// Block: PPrgArchive10

DATA_BLOCK PPrgArchive10
VERSION : 0.1
   NON_RETAIN
   VAR
      PRG : Array[901..1000] of PPrg_Data;
   END_VAR

BEGIN
   // No initialization required
END_DATA_BLOCK
